SUBAPPLICATION values_50_75_25 (* AR-Adapter-Ausgaenge fuer eine AR_AUI_MUX_3-Sollwertauswahl (K=0->OUT_50 Neutral, K=1->OUT_75, K=2->OUT_25). OUT_50 ist fest (50.0), OUT_75/OUT_25 sind proportional zum PWM_POW-Socket (0.0-1.0): bei PWM_POW=1.0 ergeben sich exakt die mit dem Multimeter kalibrierten Rohwerte 90.0/15.0 (unveraendert gegenueber der vorherigen Version mit festen Konstanten) - kleinere PWM_POW-Werte fahren proportional dazwischen, Vorbereitung fuer eine kuenftige Joystick-Ansteuerung. Name/Plug-Bezeichnungen (_75/_25) sind historisch, die tatsaechlichen kalibrierten Werte sind 90.0/15.0. *)
  (* Standard: 61499-2 *)
  (* Version 1.2, 2026-09-27, Franz Höpfinger, Meisterschulen am Ostbahnhof, Franz: 'initval_AR_75_SPAN/initval_AR_25_SPAN muessten ja beide 25 sein, nur dass wir beide korrigiert haben' - initval_AR_75_SPAN/initval_AR_25_SPAN von den bereits eingebackenen Multimeter-Werten (40.0/35.0) auf die nominelle Spanne 25.0 zurueckgesetzt, die reale Korrektur laeuft jetzt ueber 2 neue InputVars FACTOR_75/FACTOR_25 (REAL, per Parameter gesetzt) + je ein MyLib::sys::AR_R_MUL dazwischen (25.0 x FACTOR_75/_25 = 40.0/35.0 bei den bisherigen Default-Werten - unveraendertes Verhalten, nur nicht mehr eingebacken). Default-Werte in MyLib::sys::const::PWM_Konstanten::VALUES_50_75_25_FACTOR_75/_25. *)
  (* Version 1.1, 2026-09-19, Franz Höpfinger, Meisterschulen am Ostbahnhof, OUT_75/OUT_25 von festen Konstanten auf PWM_POW-proportionale Werte umgestellt (50 +/- PWM_POW*Spanne) - Vorbereitung fuer proportionale Heben/Senken-Ansteuerung per Joystick. Bei PWM_POW=1.0 unveraendert exakt die alten, mit dem Multimeter kalibrierten Rohwerte (90.0/15.0). *)
  (* Version 1.0, 2026-09-08, Franz Höpfinger, Meisterschulen am Ostbahnhof *)
  PACKAGE MyLib::sys;
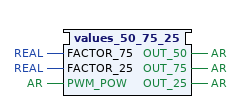
  VAR_INPUT
    FACTOR_75 : REAL := REAL#1.6; (* Multimeter-kalibrierter Korrekturfaktor auf die nominelle OUT_75-Spanne (25.0) - Default entspricht dem bisherigen eingebackenen Wert 40.0 (=25.0*1.6). Siehe MyLib::sys::const::PWM_Konstanten::VALUES_50_75_25_FACTOR_75. *)
    FACTOR_25 : REAL := REAL#1.4; (* Multimeter-kalibrierter Korrekturfaktor auf die nominelle OUT_25-Spanne (25.0) - Default entspricht dem bisherigen eingebackenen Wert 35.0 (=25.0*1.4). Siehe MyLib::sys::const::PWM_Konstanten::VALUES_50_75_25_FACTOR_25. *)
  END_VAR
  SOCKETS
    PWM_POW : adapter::types::unidirectional::AR; (* PWM Power 1.0 = Maximale Power. 0.0 Aus 0.5 Halb. *)
  END_SOCKETS
  PLUGS
    OUT_50 : adapter::types::unidirectional::AR; (* Fester Wert 50.0 (Neutral) *)
    OUT_75 : adapter::types::unidirectional::AR; (* 50.0 + PWM_POW*(25.0*FACTOR_75) - bei PWM_POW=1.0 und Default-FACTOR_75 der mit dem Multimeter kalibrierte Rohwert 90.0 *)
    OUT_25 : adapter::types::unidirectional::AR; (* 50.0 - PWM_POW*(25.0*FACTOR_25) - bei PWM_POW=1.0 und Default-FACTOR_25 der mit dem Multimeter kalibrierte Rohwert 15.0 *)
  END_PLUGS
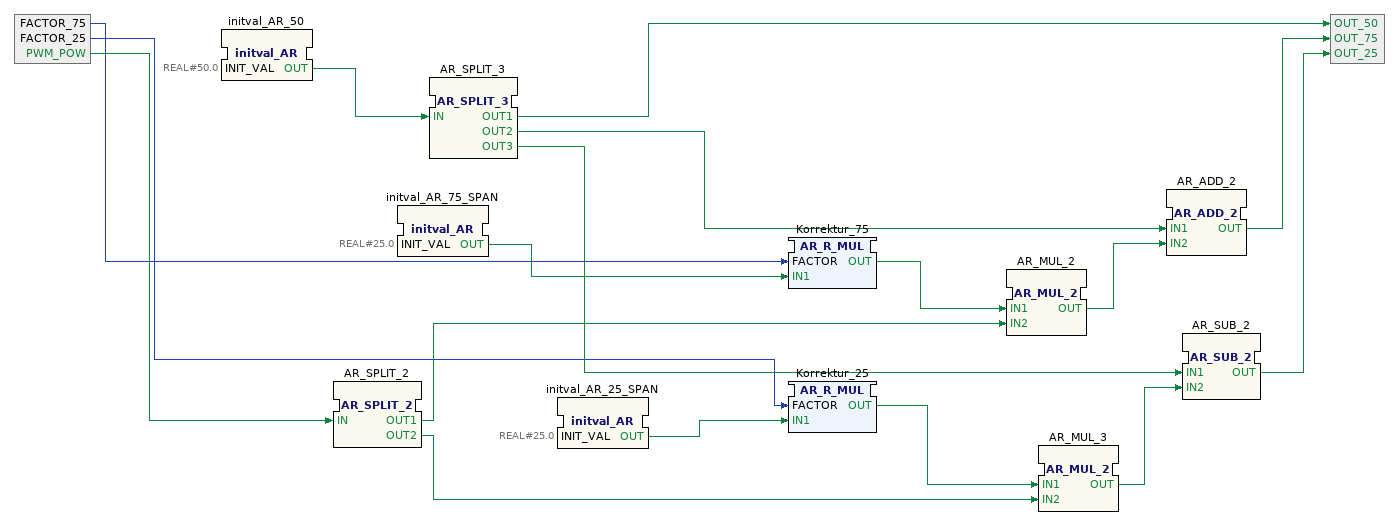
  FBS
    initval_AR_50 : adapter::types::unidirectional::AR::initval::initval_AR(INIT_VAL := REAL#50.0);
    initval_AR_75_SPAN : adapter::types::unidirectional::AR::initval::initval_AR(INIT_VAL := REAL#25.0);
    initval_AR_25_SPAN : adapter::types::unidirectional::AR::initval::initval_AR(INIT_VAL := REAL#25.0);
    AR_ADD_2 : adapter::iec61131::arithmetic::AR_ADD_2;
    AR_SUB_2 : adapter::iec61131::arithmetic::AR_SUB_2;
    AR_SPLIT_3 : adapter::events::unidirectional::AR_SPLIT_3;
    AR_MUL_2 : adapter::iec61131::arithmetic::AR_MUL_2;
    AR_MUL_3 : adapter::iec61131::arithmetic::AR_MUL_2;
    AR_SPLIT_2 : adapter::events::unidirectional::AR_SPLIT_2;
  END_FBS
  SUBAPPS
    Korrektur_75 : MyLib::sys::AR_R_MUL; (* Nominelle Spanne 25.0 x FACTOR_75 (Multimeter-Korrektur) *)
    Korrektur_25 : MyLib::sys::AR_R_MUL; (* Nominelle Spanne 25.0 x FACTOR_25 (Multimeter-Korrektur) *)
  END_SUBAPPS
  DATA_CONNECTIONS
    FACTOR_75 TO Korrektur_75.FACTOR;
    FACTOR_25 TO Korrektur_25.FACTOR;
  END_CONNECTIONS
  ADAPTER_CONNECTIONS
    AR_SPLIT_3.OUT1 TO OUT_50;
    AR_ADD_2.OUT TO OUT_75;
    AR_SUB_2.OUT TO OUT_25;
    initval_AR_50.OUT TO AR_SPLIT_3.IN;
    AR_SPLIT_3.OUT2 TO AR_ADD_2.IN1;
    initval_AR_75_SPAN.OUT TO Korrektur_75.IN1;
    Korrektur_75.OUT TO AR_MUL_2.IN1;
    AR_SPLIT_3.OUT3 TO AR_SUB_2.IN1;
    initval_AR_25_SPAN.OUT TO Korrektur_25.IN1;
    Korrektur_25.OUT TO AR_MUL_3.IN1;
    PWM_POW TO AR_SPLIT_2.IN;
    AR_MUL_2.OUT TO AR_ADD_2.IN2;
    AR_MUL_3.OUT TO AR_SUB_2.IN2;
    AR_SPLIT_2.OUT1 TO AR_MUL_2.IN2;
    AR_SPLIT_2.OUT2 TO AR_MUL_3.IN2;
  END_CONNECTIONS
END_SUBAPPLICATION
